{attribute 'qualified_only'}
VAR_GLOBAL
	ComErr, EMO_Diag,PowerIsOn AT%I*:BOOL;
	Ack,Run,Restart AT%Q*:BOOL;
END_VAR

(* stored: Version 1.1.0.1, ProductVersion 3.1.4024.10
   GVL GVL_SAFETY: Id {49aca87d-b90b-4eae-bbd2-d0dcd883e726} *)
